INTERFACE I_VisuMessage

METHOD CheckAknowledge : BOOL
VAR_INPUT
END_VAR
END_METHOD

METHOD ClearAlarmMessage : BOOL
VAR_INPUT
END_VAR
END_METHOD

METHOD ClearAllMessages : BOOL
VAR_INPUT
END_VAR
END_METHOD

METHOD ClearInfoMessage : BOOL
VAR_INPUT
END_VAR
END_METHOD

METHOD SetAlarmMessage : BOOL
VAR_INPUT
	sMessage	: STRING;
END_VAR
END_METHOD

METHOD SetErrorMessage : BOOL
VAR_INPUT
	sMessage	: STRING;
	sSequence	: STRING;
	nState		: DINT;
	nErrorCode	: DWORD;
END_VAR
END_METHOD

METHOD SetInfoMessage : BOOL
VAR_INPUT
	sMessage	: STRING;
	sSequence	: STRING;
	nState		: DINT;
END_VAR
END_METHOD

METHOD StateUpdate : BOOL
VAR_INPUT
	nState		: DINT;
	sSequence	: STRING;
END_VAR
END_METHOD

END_INTERFACE

(* stored: Version 1.1.0.1, ProductVersion 3.1.4024.13
   Itf I_VisuMessage: Id {c7fa5e2f-44b8-4fc4-8937-f550facf4207}
   Method CheckAknowledge: Id {7eed7428-3c25-41b8-98d4-2574a134fb38}
   Method ClearAlarmMessage: Id {7874348e-37eb-4e87-8833-3b0f8cd888ed}
   Method ClearAllMessages: Id {fc855211-e33d-4e48-b7ec-1d14fae18ce3}
   Method ClearInfoMessage: Id {4d665c5d-efd0-40ea-a1b2-976f6945346c}
   Method SetAlarmMessage: Id {69fcca6f-620f-458a-b038-43ef1f67b68d}
   Method SetErrorMessage: Id {e04722bf-5f2f-4613-aea8-49886abc711f}
   Method SetInfoMessage: Id {a55141da-dbff-404a-bbd9-98a0935f44a6}
   Method StateUpdate: Id {165282fe-2038-4c6a-8ff4-2a497798b3f9} *)
